{attribute 'qualified_only'}
{attribute 'no-analysis'}
{attribute 'global_init_slot' := '49992'}
VAR_GLOBAL CONSTANT
	cMaxSizeJsonDocument				: UDINT (16#FF..16#8000) 		:= 16#4000;
	cSnappyVerifyAmsNetID				: T_AmsNetID					:= TcHaxx_rplc.GCL.cLocalAmsNetId;	
	cSnappyVerifyPort					: T_SnappyVerifyPort			:= 25000;
	cSnappyVerifyInstancePath 			: STRING						:= 'TcHaxx.Snappy.Verifier.VerifyService';
	cSnappyVerifySymbol 				: STRING						:= 'Verify';
	cSnappyVerificationResultLength 	: UDINT(16#80..16#4000) 		:= 16#400;	
	cSnappyVerificationTestSuiteLength 	: UDINT(16#80..16#400) 			:= 16#100;
	cSnappyVerificationTestNameLength 	: UDINT(16#80..16#400) 			:= 16#100;			
END_VAR

(* stored: Version 1.1.0.1, ProductVersion 3.1.4026.18
   GVL Param_TcHaxx_Snappy: Id {9fb7b88a-4b4f-41ab-b59b-8ee6e4c3fd80}, ParameterList True *)
